TYPE E_WashState :
(
    Idle,
    Filling,
    Washing,
    Draining,
    Completed
);
END_TYPE

(* stored: Version 1.1.0.1, ProductVersion 3.1.4024.16
   DUT E_WashState: Id {34307ab2-1eb6-46f9-9ffb-edd66d850057} *)
